// TIA Portal V17 export
// export: Created 2026-04-12T10:31:32.2362113Z, ExportSetting WithDefaults, DisplayName Totally Integrated Automation Portal, DisplayVersion V17 Update 4, DisplayName TIA Portal Openness, DisplayVersion V17 Update 4, DisplayName TIA Portal Version Control Interface, DisplayVersion V17, DisplayName SINAMICS Startdrive Advanced, DisplayVersion V17, DisplayName SINAMICS Startdrive G130, G150, S120, S150, SINAMICS MV, S210, DisplayVersion V17, DisplayName SINAMICS Startdrive G110M, G120, G120C, G120D, G120P, G115D, DisplayVersion V17, DisplayName STEP 7 Professional, DisplayVersion V17 Update 4, DisplayName STEP 7 Safety, DisplayVersion V17, DisplayName WinCC Advanced, DisplayVersion V17 Update 4
FUNCTION "输入信号转换块" : Void   // FC2, LAD
{ S7_Optimized_Access := 'TRUE' }
VERSION : 0.1
// stored: AutoNumber false, IsIECCheckEnabled false, SetENOAutomatically false, UDAEnableTagReadback false
BEGIN

REGION Network 1: 1区-8输入信号
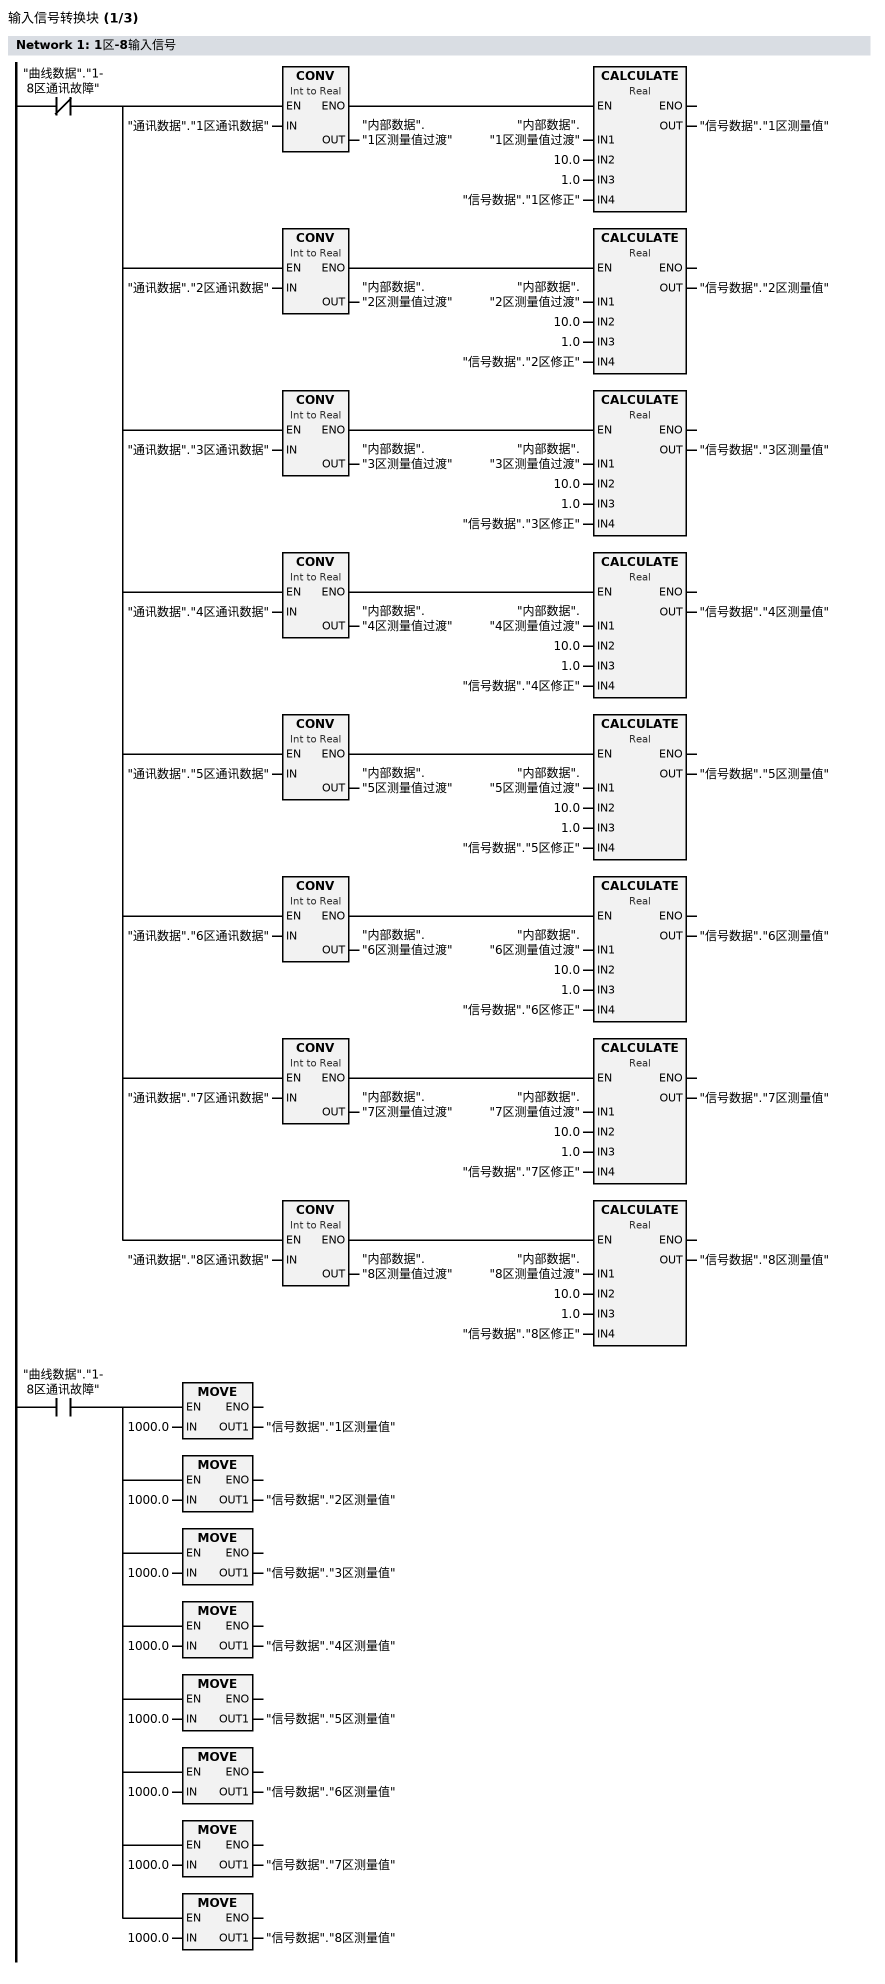
   RUNG wire#powerrail
      I_Contact( "曲线数据"."1-8区通讯故障" )
      wire#w1
      { S7_Templates := "[SrcType := Int, DestType := Real]" } Convert(in := "通讯数据"."1区通讯数据", out => "内部数据"."1区测量值过渡")
      { S7_Templates := "SrcType := Real"; S7_Expression := "IN1/IN2*IN3-IN4" } Calculate(in1 := "内部数据"."1区测量值过渡", in2 := 10.0, in3 := 1.0, in4 := "信号数据"."1区修正", out => "信号数据"."1区测量值")
   END_RUNG
   RUNG wire#w1
      { S7_Templates := "[SrcType := Int, DestType := Real]" } Convert(in := "通讯数据"."2区通讯数据", out => "内部数据"."2区测量值过渡")
      { S7_Templates := "SrcType := Real"; S7_Expression := "IN1/IN2*IN3-IN4" } Calculate(in1 := "内部数据"."2区测量值过渡", in2 := 10.0, in3 := 1.0, in4 := "信号数据"."2区修正", out => "信号数据"."2区测量值")
   END_RUNG
   RUNG wire#w1
      { S7_Templates := "[SrcType := Int, DestType := Real]" } Convert(in := "通讯数据"."3区通讯数据", out => "内部数据"."3区测量值过渡")
      { S7_Templates := "SrcType := Real"; S7_Expression := "IN1/IN2*IN3-IN4" } Calculate(in1 := "内部数据"."3区测量值过渡", in2 := 10.0, in3 := 1.0, in4 := "信号数据"."3区修正", out => "信号数据"."3区测量值")
   END_RUNG
   RUNG wire#w1
      { S7_Templates := "[SrcType := Int, DestType := Real]" } Convert(in := "通讯数据"."4区通讯数据", out => "内部数据"."4区测量值过渡")
      { S7_Templates := "SrcType := Real"; S7_Expression := "IN1/IN2*IN3-IN4" } Calculate(in1 := "内部数据"."4区测量值过渡", in2 := 10.0, in3 := 1.0, in4 := "信号数据"."4区修正", out => "信号数据"."4区测量值")
   END_RUNG
   RUNG wire#w1
      { S7_Templates := "[SrcType := Int, DestType := Real]" } Convert(in := "通讯数据"."5区通讯数据", out => "内部数据"."5区测量值过渡")
      { S7_Templates := "SrcType := Real"; S7_Expression := "IN1/IN2*IN3-IN4" } Calculate(in1 := "内部数据"."5区测量值过渡", in2 := 10.0, in3 := 1.0, in4 := "信号数据"."5区修正", out => "信号数据"."5区测量值")
   END_RUNG
   RUNG wire#w1
      { S7_Templates := "[SrcType := Int, DestType := Real]" } Convert(in := "通讯数据"."6区通讯数据", out => "内部数据"."6区测量值过渡")
      { S7_Templates := "SrcType := Real"; S7_Expression := "IN1/IN2*IN3-IN4" } Calculate(in1 := "内部数据"."6区测量值过渡", in2 := 10.0, in3 := 1.0, in4 := "信号数据"."6区修正", out => "信号数据"."6区测量值")
   END_RUNG
   RUNG wire#w1
      { S7_Templates := "[SrcType := Int, DestType := Real]" } Convert(in := "通讯数据"."7区通讯数据", out => "内部数据"."7区测量值过渡")
      { S7_Templates := "SrcType := Real"; S7_Expression := "IN1/IN2*IN3-IN4" } Calculate(in1 := "内部数据"."7区测量值过渡", in2 := 10.0, in3 := 1.0, in4 := "信号数据"."7区修正", out => "信号数据"."7区测量值")
   END_RUNG
   RUNG wire#w1
      { S7_Templates := "[SrcType := Int, DestType := Real]" } Convert(in := "通讯数据"."8区通讯数据", out => "内部数据"."8区测量值过渡")
      { S7_Templates := "SrcType := Real"; S7_Expression := "IN1/IN2*IN3-IN4" } Calculate(in1 := "内部数据"."8区测量值过渡", in2 := 10.0, in3 := 1.0, in4 := "信号数据"."8区修正", out => "信号数据"."8区测量值")
   END_RUNG
   RUNG wire#powerrail
      Contact( "曲线数据"."1-8区通讯故障" )
      wire#w2
      Move(in := 1000.0, out1 => "信号数据"."1区测量值")
   END_RUNG
   RUNG wire#w2
      Move(in := 1000.0, out1 => "信号数据"."2区测量值")
   END_RUNG
   RUNG wire#w2
      Move(in := 1000.0, out1 => "信号数据"."3区测量值")
   END_RUNG
   RUNG wire#w2
      Move(in := 1000.0, out1 => "信号数据"."4区测量值")
   END_RUNG
   RUNG wire#w2
      Move(in := 1000.0, out1 => "信号数据"."5区测量值")
   END_RUNG
   RUNG wire#w2
      Move(in := 1000.0, out1 => "信号数据"."6区测量值")
   END_RUNG
   RUNG wire#w2
      Move(in := 1000.0, out1 => "信号数据"."7区测量值")
   END_RUNG
   RUNG wire#w2
      Move(in := 1000.0, out1 => "信号数据"."8区测量值")
   END_RUNG
   // the same network as SCL:
   IF NOT "曲线数据"."1-8区通讯故障" THEN
       "内部数据"."1区测量值过渡" := INT_TO_REAL("通讯数据"."1区通讯数据");
       "信号数据"."1区测量值" := "内部数据"."1区测量值过渡"/10.0*1.0-"信号数据"."1区修正";
       "内部数据"."2区测量值过渡" := INT_TO_REAL("通讯数据"."2区通讯数据");
       "信号数据"."2区测量值" := "内部数据"."2区测量值过渡"/10.0*1.0-"信号数据"."2区修正";
       "内部数据"."3区测量值过渡" := INT_TO_REAL("通讯数据"."3区通讯数据");
       "信号数据"."3区测量值" := "内部数据"."3区测量值过渡"/10.0*1.0-"信号数据"."3区修正";
       "内部数据"."4区测量值过渡" := INT_TO_REAL("通讯数据"."4区通讯数据");
       "信号数据"."4区测量值" := "内部数据"."4区测量值过渡"/10.0*1.0-"信号数据"."4区修正";
       "内部数据"."5区测量值过渡" := INT_TO_REAL("通讯数据"."5区通讯数据");
       "信号数据"."5区测量值" := "内部数据"."5区测量值过渡"/10.0*1.0-"信号数据"."5区修正";
       "内部数据"."6区测量值过渡" := INT_TO_REAL("通讯数据"."6区通讯数据");
       "信号数据"."6区测量值" := "内部数据"."6区测量值过渡"/10.0*1.0-"信号数据"."6区修正";
       "内部数据"."7区测量值过渡" := INT_TO_REAL("通讯数据"."7区通讯数据");
       "信号数据"."7区测量值" := "内部数据"."7区测量值过渡"/10.0*1.0-"信号数据"."7区修正";
       "内部数据"."8区测量值过渡" := INT_TO_REAL("通讯数据"."8区通讯数据");
       "信号数据"."8区测量值" := "内部数据"."8区测量值过渡"/10.0*1.0-"信号数据"."8区修正";
   END_IF;
   IF "曲线数据"."1-8区通讯故障" THEN
       "信号数据"."1区测量值" := 1000.0;
       "信号数据"."2区测量值" := 1000.0;
       "信号数据"."3区测量值" := 1000.0;
       "信号数据"."4区测量值" := 1000.0;
       "信号数据"."5区测量值" := 1000.0;
       "信号数据"."6区测量值" := 1000.0;
       "信号数据"."7区测量值" := 1000.0;
       "信号数据"."8区测量值" := 1000.0;
   END_IF;
END_REGION

REGION Network 2: 9区-15区输入信号
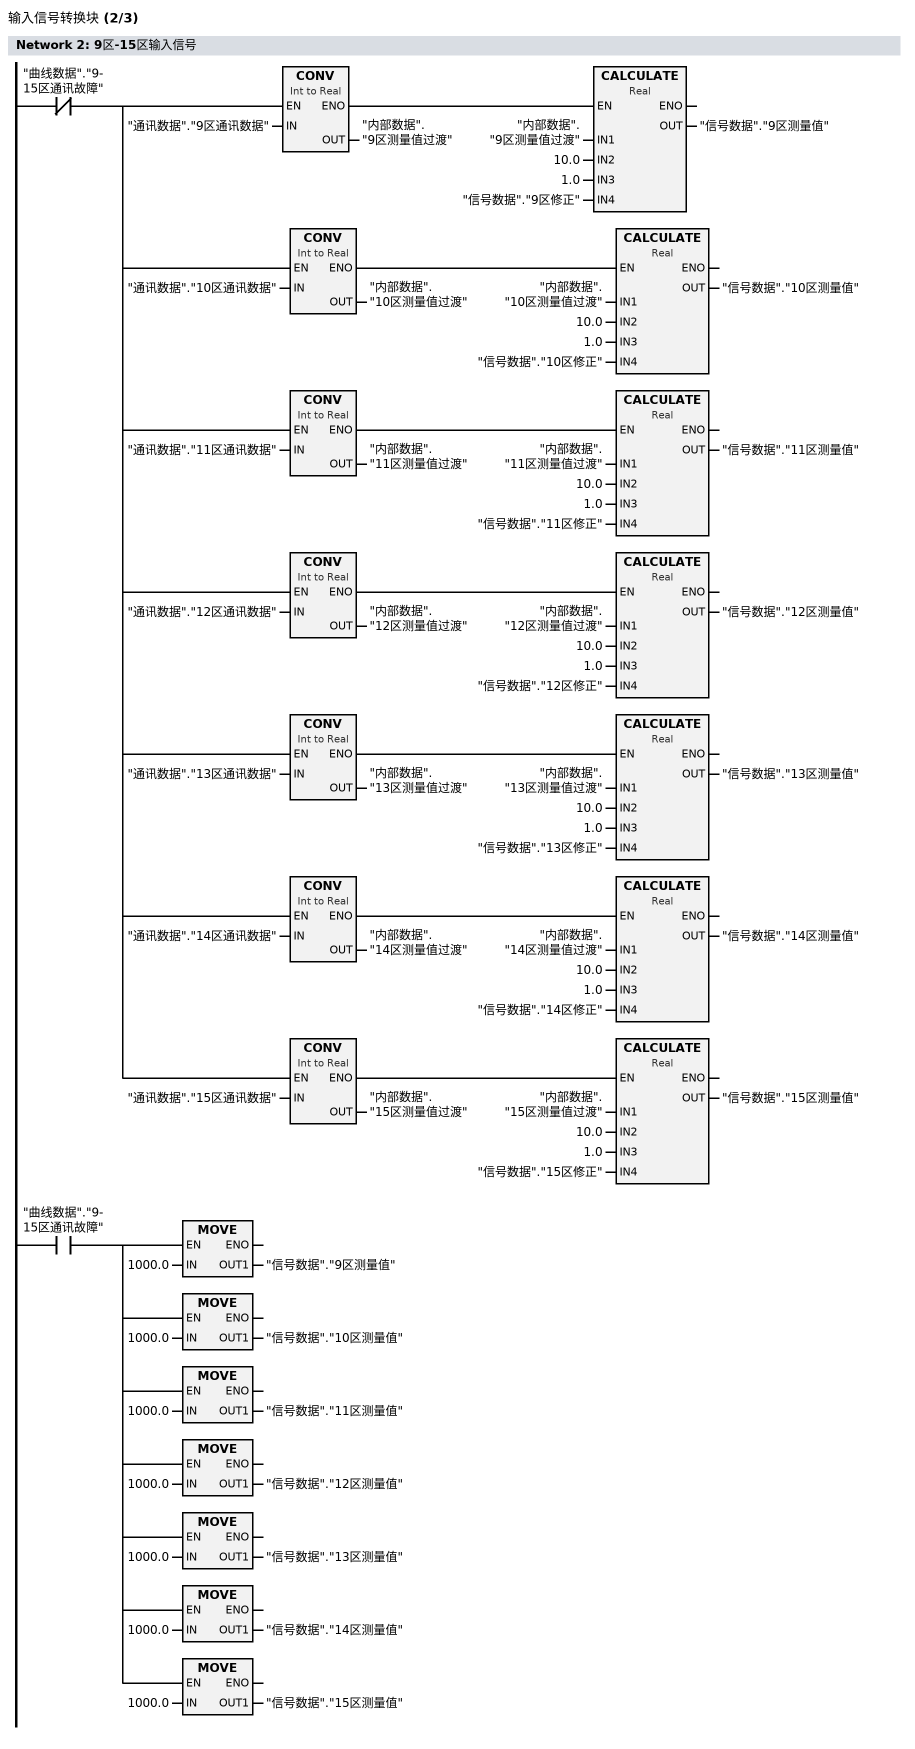
   RUNG wire#powerrail
      I_Contact( "曲线数据"."9-15区通讯故障" )
      wire#w1
      { S7_Templates := "[SrcType := Int, DestType := Real]" } Convert(in := "通讯数据"."9区通讯数据", out => "内部数据"."9区测量值过渡")
      { S7_Templates := "SrcType := Real"; S7_Expression := "IN1/IN2*IN3-IN4" } Calculate(in1 := "内部数据"."9区测量值过渡", in2 := 10.0, in3 := 1.0, in4 := "信号数据"."9区修正", out => "信号数据"."9区测量值")
   END_RUNG
   RUNG wire#w1
      { S7_Templates := "[SrcType := Int, DestType := Real]" } Convert(in := "通讯数据"."10区通讯数据", out => "内部数据"."10区测量值过渡")
      { S7_Templates := "SrcType := Real"; S7_Expression := "IN1/IN2*IN3-IN4" } Calculate(in1 := "内部数据"."10区测量值过渡", in2 := 10.0, in3 := 1.0, in4 := "信号数据"."10区修正", out => "信号数据"."10区测量值")
   END_RUNG
   RUNG wire#w1
      { S7_Templates := "[SrcType := Int, DestType := Real]" } Convert(in := "通讯数据"."11区通讯数据", out => "内部数据"."11区测量值过渡")
      { S7_Templates := "SrcType := Real"; S7_Expression := "IN1/IN2*IN3-IN4" } Calculate(in1 := "内部数据"."11区测量值过渡", in2 := 10.0, in3 := 1.0, in4 := "信号数据"."11区修正", out => "信号数据"."11区测量值")
   END_RUNG
   RUNG wire#w1
      { S7_Templates := "[SrcType := Int, DestType := Real]" } Convert(in := "通讯数据"."12区通讯数据", out => "内部数据"."12区测量值过渡")
      { S7_Templates := "SrcType := Real"; S7_Expression := "IN1/IN2*IN3-IN4" } Calculate(in1 := "内部数据"."12区测量值过渡", in2 := 10.0, in3 := 1.0, in4 := "信号数据"."12区修正", out => "信号数据"."12区测量值")
   END_RUNG
   RUNG wire#w1
      { S7_Templates := "[SrcType := Int, DestType := Real]" } Convert(in := "通讯数据"."13区通讯数据", out => "内部数据"."13区测量值过渡")
      { S7_Templates := "SrcType := Real"; S7_Expression := "IN1/IN2*IN3-IN4" } Calculate(in1 := "内部数据"."13区测量值过渡", in2 := 10.0, in3 := 1.0, in4 := "信号数据"."13区修正", out => "信号数据"."13区测量值")
   END_RUNG
   RUNG wire#w1
      { S7_Templates := "[SrcType := Int, DestType := Real]" } Convert(in := "通讯数据"."14区通讯数据", out => "内部数据"."14区测量值过渡")
      { S7_Templates := "SrcType := Real"; S7_Expression := "IN1/IN2*IN3-IN4" } Calculate(in1 := "内部数据"."14区测量值过渡", in2 := 10.0, in3 := 1.0, in4 := "信号数据"."14区修正", out => "信号数据"."14区测量值")
   END_RUNG
   RUNG wire#w1
      { S7_Templates := "[SrcType := Int, DestType := Real]" } Convert(in := "通讯数据"."15区通讯数据", out => "内部数据"."15区测量值过渡")
      { S7_Templates := "SrcType := Real"; S7_Expression := "IN1/IN2*IN3-IN4" } Calculate(in1 := "内部数据"."15区测量值过渡", in2 := 10.0, in3 := 1.0, in4 := "信号数据"."15区修正", out => "信号数据"."15区测量值")
   END_RUNG
   RUNG wire#powerrail
      Contact( "曲线数据"."9-15区通讯故障" )
      wire#w2
      Move(in := 1000.0, out1 => "信号数据"."9区测量值")
   END_RUNG
   RUNG wire#w2
      Move(in := 1000.0, out1 => "信号数据"."10区测量值")
   END_RUNG
   RUNG wire#w2
      Move(in := 1000.0, out1 => "信号数据"."11区测量值")
   END_RUNG
   RUNG wire#w2
      Move(in := 1000.0, out1 => "信号数据"."12区测量值")
   END_RUNG
   RUNG wire#w2
      Move(in := 1000.0, out1 => "信号数据"."13区测量值")
   END_RUNG
   RUNG wire#w2
      Move(in := 1000.0, out1 => "信号数据"."14区测量值")
   END_RUNG
   RUNG wire#w2
      Move(in := 1000.0, out1 => "信号数据"."15区测量值")
   END_RUNG
   // the same network as SCL:
   IF NOT "曲线数据"."9-15区通讯故障" THEN
       "内部数据"."9区测量值过渡" := INT_TO_REAL("通讯数据"."9区通讯数据");
       "信号数据"."9区测量值" := "内部数据"."9区测量值过渡"/10.0*1.0-"信号数据"."9区修正";
       "内部数据"."10区测量值过渡" := INT_TO_REAL("通讯数据"."10区通讯数据");
       "信号数据"."10区测量值" := "内部数据"."10区测量值过渡"/10.0*1.0-"信号数据"."10区修正";
       "内部数据"."11区测量值过渡" := INT_TO_REAL("通讯数据"."11区通讯数据");
       "信号数据"."11区测量值" := "内部数据"."11区测量值过渡"/10.0*1.0-"信号数据"."11区修正";
       "内部数据"."12区测量值过渡" := INT_TO_REAL("通讯数据"."12区通讯数据");
       "信号数据"."12区测量值" := "内部数据"."12区测量值过渡"/10.0*1.0-"信号数据"."12区修正";
       "内部数据"."13区测量值过渡" := INT_TO_REAL("通讯数据"."13区通讯数据");
       "信号数据"."13区测量值" := "内部数据"."13区测量值过渡"/10.0*1.0-"信号数据"."13区修正";
       "内部数据"."14区测量值过渡" := INT_TO_REAL("通讯数据"."14区通讯数据");
       "信号数据"."14区测量值" := "内部数据"."14区测量值过渡"/10.0*1.0-"信号数据"."14区修正";
       "内部数据"."15区测量值过渡" := INT_TO_REAL("通讯数据"."15区通讯数据");
       "信号数据"."15区测量值" := "内部数据"."15区测量值过渡"/10.0*1.0-"信号数据"."15区修正";
   END_IF;
   IF "曲线数据"."9-15区通讯故障" THEN
       "信号数据"."9区测量值" := 1000.0;
       "信号数据"."10区测量值" := 1000.0;
       "信号数据"."11区测量值" := 1000.0;
       "信号数据"."12区测量值" := 1000.0;
       "信号数据"."13区测量值" := 1000.0;
       "信号数据"."14区测量值" := 1000.0;
       "信号数据"."15区测量值" := 1000.0;
   END_IF;
END_REGION

REGION Network 3: 风压输入信号
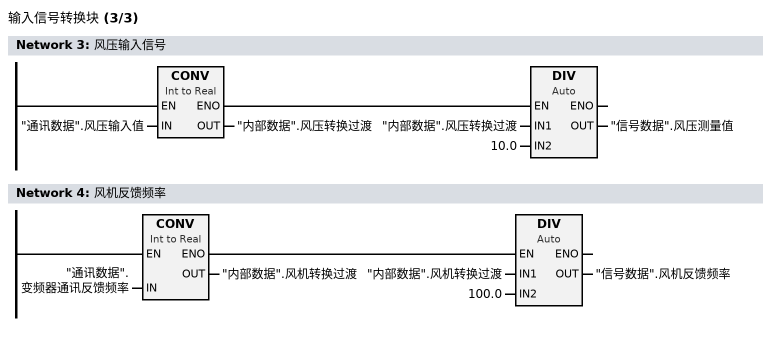
   RUNG wire#powerrail
      { S7_Templates := "[SrcType := Int, DestType := Real]" } Convert(in := "通讯数据".风压输入值, out => "内部数据".风压转换过渡)
      Div(in1 := "内部数据".风压转换过渡, in2 := 10.0, out => "信号数据".风压测量值)
   END_RUNG
   // the same network as SCL:
   "内部数据".风压转换过渡 := INT_TO_REAL("通讯数据".风压输入值);
   "信号数据".风压测量值 := "内部数据".风压转换过渡 / 10.0;
END_REGION

REGION Network 4: 风机反馈频率
   RUNG wire#powerrail
      { S7_Templates := "[SrcType := Int, DestType := Real]" } Convert(in := "通讯数据".变频器通讯反馈频率, out => "内部数据".风机转换过渡)
      Div(in1 := "内部数据".风机转换过渡, in2 := 100.0, out => "信号数据".风机反馈频率)
   END_RUNG
   // the same network as SCL:
   "内部数据".风机转换过渡 := INT_TO_REAL("通讯数据".变频器通讯反馈频率);
   "信号数据".风机反馈频率 := "内部数据".风机转换过渡 / 100.0;
END_REGION
END_FUNCTION
